{attribute 'GeneratedUsingTerminal: EP7402-0057-0017'}
{attribute addProperty BoxType "EP7402-0057-0017"}
{attribute addProperty Id "VelocityAT %Q*INT2AccellerationAT %Q*UINT2DeccelerationAT %Q*UINT2"}
{attribute addProperty CRC "3869082405"}
{attribute addProperty Size "6"}
TYPE STM_Target_Velocity_Channel_E69D8325 EXTENDS OutputBase_10CEE7DE :
STRUCT
	{attribute addProperty Name "Velocity"}
	Velocity AT %Q* : INT;
	{attribute addProperty Name "Accelleration"}
	Accelleration AT %Q* : UINT;
	{attribute addProperty Name "Decceleration"}
	Decceleration AT %Q* : UINT;
END_STRUCT
END_TYPE

(* stored: Version 1.2.0.0, ProductVersion 3.1.4024.11
   DUT STM_Target_Velocity_Channel_E69D8325: Id {8d64b44d-8224-4448-81e7-80e54f14124f} *)
